(* IEC 61131-3 sources: StewartPlatform/Class/IONet, 1 file *)

(* ---- IONet.st ---- *)
(*!
<Class
	Name               = "IONet"
	Revision           = "0.0"
	RealtimeTask       = "false"
	CyclicTask         = "true"
	DefCyclictime      = "10 ms"
	BackgroundTask     = "false"
	Sigmatek           = "false"
	OSInterface        = "false"
	HighPriority       = "false"
	Automatic          = "false"
	UpdateMode         = "Prescan"
	SharedCommandTable = "true"
	Objectsize         = "(720,360)">
	<Channels>
		<Server Name="ClassSvr" Visualized="false" Initialize="false" WriteProtected="true" Retentive="false"/>
		<Server Name="Counter1" Visualized="false" Initialize="true" DefValue="2000" WriteProtected="false" Retentive="File"/>
		<Server Name="Counter2" Visualized="false" Initialize="true" DefValue="8000" WriteProtected="false" Retentive="File"/>
		<Server Name="Counter3" Visualized="false" Initialize="true" DefValue="5000" WriteProtected="false" Retentive="File"/>
		<Server Name="DefaultSpeed" Visualized="false" Initialize="false" WriteProtected="false" Retentive="File"/>
		<Server Name="diff" Visualized="false" Initialize="false" WriteProtected="false" Retentive="File"/>
		<Server Name="Direction1" Visualized="false" Initialize="true" DefValue="0" WriteProtected="false" Retentive="File"/>
		<Server Name="Direction2" Visualized="false" Initialize="true" DefValue="1" WriteProtected="false" Retentive="File"/>
		<Server Name="Direction3" Visualized="false" Initialize="true" DefValue="0" WriteProtected="false" Retentive="File"/>
		<Server Name="DropDownSpeed" Visualized="false" Initialize="false" WriteProtected="false" Retentive="File"/>
		<Server Name="Error1" Visualized="false" Initialize="false" WriteProtected="false" Retentive="File"/>
		<Server Name="Error2" Visualized="false" Initialize="false" WriteProtected="false" Retentive="File"/>
		<Server Name="Error3" Visualized="false" Initialize="false" WriteProtected="false" Retentive="File"/>
		<Server Name="Error4" Visualized="false" Initialize="false" WriteProtected="false" Retentive="File"/>
		<Server Name="Error5" Visualized="false" Initialize="false" WriteProtected="false" Retentive="File"/>
		<Server Name="Error6" Visualized="false" Initialize="false" WriteProtected="false" Retentive="File"/>
		<Server Name="InitCounter1" Visualized="false" Initialize="false" WriteProtected="false" Retentive="File"/>
		<Server Name="InitialTolerance" Visualized="false" Initialize="false" WriteProtected="false" Retentive="File"/>
		<Server Name="Integrator1" Visualized="false" Initialize="false" WriteProtected="false" Retentive="File"/>
		<Server Name="Integrator2" Visualized="false" Initialize="false" WriteProtected="false" Retentive="File"/>
		<Server Name="Integrator3" Visualized="false" Initialize="false" WriteProtected="false" Retentive="File"/>
		<Server Name="Integrator4" Visualized="false" Initialize="false" WriteProtected="false" Retentive="File"/>
		<Server Name="Integrator5" Visualized="false" Initialize="false" WriteProtected="false" Retentive="File"/>
		<Server Name="Integrator6" Visualized="false" Initialize="false" WriteProtected="false" Retentive="File"/>
		<Server Name="Kd" Visualized="false" Initialize="true" DefValue="0" WriteProtected="false" Retentive="File"/>
		<Server Name="Ki" Visualized="false" Initialize="false" WriteProtected="false" Retentive="File"/>
		<Server Name="Kp" Visualized="false" Initialize="true" DefValue="5" WriteProtected="false" Retentive="File"/>
		<Server Name="LowerLimit" Visualized="false" Initialize="false" WriteProtected="false" Retentive="File"/>
		<Server Name="Mode" Visualized="false" Initialize="false" WriteProtected="false" Retentive="File"/>
		<Server Name="ModeDoneCounter" Visualized="false" Initialize="false" WriteProtected="true" Retentive="false"/>
		<Server Name="ModeDoneSmoother" Visualized="false" Initialize="false" WriteProtected="false" Retentive="File"/>
		<Server Name="Phase" Visualized="false" Initialize="false" WriteProtected="false" Retentive="File"/>
		<Server Name="Prior_error1" Visualized="false" Initialize="false" WriteProtected="false" Retentive="File"/>
		<Server Name="Prior_error2" Visualized="false" Initialize="false" WriteProtected="false" Retentive="File"/>
		<Server Name="Prior_error3" Visualized="false" Initialize="false" WriteProtected="false" Retentive="File"/>
		<Server Name="Prior_error4" Visualized="false" Initialize="false" WriteProtected="false" Retentive="File"/>
		<Server Name="Prior_error5" Visualized="false" Initialize="false" WriteProtected="false" Retentive="File"/>
		<Server Name="Prior_error6" Visualized="false" Initialize="false" WriteProtected="false" Retentive="File"/>
		<Server Name="Speed" Visualized="false" Initialize="false" WriteProtected="false" Retentive="File"/>
		<Server Name="System_state" Visualized="false" Initialize="false" WriteProtected="false" Retentive="File"/>
		<Server Name="UpperLimit" Visualized="false" Initialize="false" WriteProtected="false" Retentive="File"/>
		<Client Name="EnableCircuit" Required="true" Internal="false"/>
		<Client Name="ExternalController" Required="true" Internal="false"/>
		<Client Name="I1" Required="true" Internal="false"/>
		<Client Name="I2" Required="true" Internal="false"/>
		<Client Name="I3" Required="true" Internal="false"/>
		<Client Name="I4" Required="true" Internal="false"/>
		<Client Name="I5" Required="true" Internal="false"/>
		<Client Name="I6" Required="true" Internal="false"/>
		<Client Name="O1" Required="true" Internal="false"/>
		<Client Name="O2" Required="true" Internal="false"/>
		<Client Name="O3" Required="true" Internal="false"/>
		<Client Name="O4" Required="true" Internal="false"/>
		<Client Name="O5" Required="true" Internal="false"/>
		<Client Name="O6" Required="true" Internal="false"/>
		<Client Name="Pressurize" Required="true" Internal="false"/>
		<Client Name="ResetButton" Required="true" Internal="false"/>
		<Client Name="ResetButtonLamp" Required="true" Internal="false"/>
		<Client Name="ResetEStop" Required="true" Internal="false"/>
		<Client Name="StartButton" Required="true" Internal="false"/>
		<Client Name="StartButtonLamp" Required="true" Internal="false"/>
		<Client Name="StartPumps" Required="true" Internal="false"/>
		<Client Name="StopButton" Required="true" Internal="false"/>
		<Client Name="StopButtonLamp" Required="true" Internal="false"/>
		<Client Name="SystemEnable" Required="true" Internal="false"/>
		<Client Name="SystemOKLamp" Required="true" Internal="false"/>
	</Channels>
</Class>
*)
IONet : CLASS
  //Servers:
	ClassSvr 	: SvrChCmd_DINT;
	Counter1 	: SvrCh_DINT;
	Counter2 	: SvrCh_DINT;
	Counter3 	: SvrCh_DINT;
	InitCounter1 	: SvrCh_DINT;
	Direction1 	: SvrCh_UDINT;
	Direction2 	: SvrCh_DINT;
	Direction3 	: SvrCh_DINT;
	Kp 	: SvrCh_DINT;
	Kd 	: SvrCh_DINT;
	Ki 	: SvrCh_DINT;
	Mode 	: SvrCh_DINT;
	Phase 	: SvrCh_DINT;
	System_state 	: SvrCh_DINT;
	Speed 	: SvrCh_DINT;
	DropDownSpeed 	: SvrCh_DINT;
	DefaultSpeed 	: SvrCh_DINT;
	Prior_error1 	: SvrCh_DINT;
	Prior_error2 	: SvrCh_DINT;
	Prior_error3 	: SvrCh_DINT;
	Prior_error4 	: SvrCh_DINT;
	Prior_error5 	: SvrCh_DINT;
	Prior_error6 	: SvrCh_DINT;
	Error1 	: SvrCh_DINT;
	Error2 	: SvrCh_DINT;
	Error3 	: SvrCh_DINT;
	Error4 	: SvrCh_DINT;
	Error5 	: SvrCh_DINT;
	Error6 	: SvrCh_DINT;
	Integrator1 	: SvrCh_DINT;
	Integrator2 	: SvrCh_DINT;
	Integrator3 	: SvrCh_DINT;
	Integrator4 	: SvrCh_DINT;
	Integrator5 	: SvrCh_DINT;
	Integrator6 	: SvrCh_DINT;
	LowerLimit 	: SvrCh_DINT;
	UpperLimit 	: SvrCh_DINT;
	diff 	: SvrCh_DINT;
	InitialTolerance 	: SvrCh_DINT;
	ModeDoneSmoother 	: SvrCh_DINT;
	ModeDoneCounter 	: SvrCh_DINT;
  //Clients:
	StartButton 	: CltCh_DINT;
	StartButtonLamp 	: CltCh_DINT;
	StopButton 	: CltCh_DINT;
	StopButtonLamp 	: CltCh_DINT;
	ResetButton 	: CltCh_DINT;
	ResetButtonLamp 	: CltCh_DINT;
	SystemEnable 	: CltCh_DINT;
	EnableCircuit 	: CltCh_DINT;
	SystemOKLamp 	: CltCh_DINT;
	StartPumps 	: CltCh_DINT;
	Pressurize 	: CltCh_DINT;
	ResetEStop 	: CltCh_DINT;
	ExternalController 	: CltCh_DINT;
	O1 	: CltCh_DINT;
	O2 	: CltCh_DINT;
	O3 	: CltCh_DINT;
	O4 	: CltCh_DINT;
	O5 	: CltCh_DINT;
	O6 	: CltCh_DINT;
	I1 	: CltCh_DINT;
	I2 	: CltCh_DINT;
	I3 	: CltCh_DINT;
	I4 	: CltCh_DINT;
	I5 	: CltCh_DINT;
	I6 	: CltCh_DINT;
  //Variables:
  //Functions:

	FUNCTION VIRTUAL GLOBAL Init;

	FUNCTION VIRTUAL GLOBAL CyWork
		VAR_INPUT
			EAX 	: UDINT;
		END_VAR
		VAR_OUTPUT
			state (EAX) 	: UDINT;
		END_VAR;

	FUNCTION LimitOutput
		VAR_INPUT
			unlimited_output 	: DINT;
		END_VAR
		VAR_OUTPUT
			limited_output 	: DINT;
		END_VAR;

	FUNCTION UpdateMode;

	FUNCTION InitializeCounters;

	FUNCTION UpdateCounters;

	FUNCTION DecreaseCounters;

	FUNCTION CylRef
		VAR_INPUT
			cyl 	: DINT;
		END_VAR
		VAR_OUTPUT
			ref 	: DINT;
		END_VAR;

	FUNCTION GoToInitial
		VAR_INPUT
			ref 	: DINT;
			actual 	: DINT;
		END_VAR
		VAR_OUTPUT
			newref 	: DINT;
		END_VAR;

	FUNCTION ResetPriorErrors;

	FUNCTION SetPriorErrors;

	FUNCTION ResetIntegrators;

	FUNCTION UpdateIntegrators;

	FUNCTION InitializeMode;

	FUNCTION AbsoluteValue
		VAR_INPUT
			Actual 	: DINT;
		END_VAR
		VAR_OUTPUT
			Absolute 	: DINT;
		END_VAR;
  //Tables:
	FUNCTION @STD
		VAR_OUTPUT
			ret_code	: CONFSTATES;
		END_VAR;
	FUNCTION GLOBAL TAB @CT_;
END_CLASS;

FUNCTION VIRTUAL GLOBAL IONet::Init
  if _FirstScan then
    Kp := 5;
    Kd := 20;
    Ki := 1;
    LowerLimit := 500;        // Lowest reachable point of cylinders
    Direction1 := 0;
    Direction2 := 0;
    Direction3 := 0;
    Counter1 := LowerLimit;
    Counter2 := LowerLimit;
    Counter3 := LowerLimit;
    DefaultSpeed := 6;        // Speed with which to increase counters every 10ms
    InitialTolerance := 300;  // Tolerance to initial mode position below which the mode is started
    DropDownSpeed := 10;      // Speed to drop down with when stop button is pressed
    System_state := 0;        // System state: 0 = SAFETY, 1 = ON, 2 = IDLE, 3 = PAUSED
    // SAFETY: a safety reset is required to go to System_state IDLE
    // ON: system is doing a sequence of movements
    // IDLE: System slowly moves to lowest position and stays there (controlled by buttons)
    // PAUSED: System slowly moves to lowest position and stays there (controlled by external controller)
    Mode := 1;                // Mode indicates which movement to perform
    ModeDoneSmoother := 50;   // To let the platform stabilize before starting next mode
    ModeDoneCounter := 0;
    Phase := 1;               // Phase indicates the part of the mode we are in (1 = go to initial, 2 = outbound, 3 = inbound, 4 = done)
    // Mode 1: up-down Z-direction (cylinder 1-6 use direction1 and counter1)
    // Mode 2: rotate yaw (cylinder 1,3,5 use direction1 and counter1, others use direction2 and counter2)
    // Mode 3: simultaneous roll-pitch (cylinder 1&6 use direction1 and counter1, cylinder 2&3 use direction2 and counter2, others use direction3 and counter3)
    // Mode 4: planar x-y direction TODO
    ResetPriorErrors();       // Reset prior errors for derivative control action
    ResetIntegrators();       // Reset integrators for integral control action
  end_if;

END_FUNCTION

FUNCTION VIRTUAL GLOBAL IONet::CyWork
	VAR_INPUT
		EAX 	: UDINT;
	END_VAR
	VAR_OUTPUT
		state (EAX) 	: UDINT;
	END_VAR

  // Read all inputs
	StartButton := StartButton.Read();
	StopButton := StopButton.Read();
	ResetButton := ResetButton.Read();
  SystemEnable := SystemEnable.Read(); // Safety circuit input
  ExternalController := ExternalController.Read(); // External controller
  I1 := I1.Read();
  I2 := I2.Read();
  I3 := I3.Read();
  I4 := I4.Read();
  I5 := I5.Read();
  I6 := I6.Read();

  // If safety circuit is OK, enable circuit and pumps
  // THIS CHECK SHOULD ALWAYS BE AT THE BEGINNING OF THE LOOP
  // ***************************************
  if SystemEnable = 1 then
    SystemOKLamp := 1;
    EnableCircuit := 1;
    StartPumps := 1;
    // TODO: pressure low should prevent system from falling down but this does not work currently
    Pressurize := 1; // no outwards cylinder movement when 0
  else
    // Set state variables
    System_state := 0;      // System state SAFETY
    Mode := 1;              // Mode starts at 1 again
    InitializeMode();       // Re-initialize mode
    ResetPriorErrors();     // Reset prior errors for derivative control action
    ResetIntegrators();     // Reset integrators for integral control action
    // Turn everything off
    ResetEStop := 0;
    SystemOKLamp := 0;
    EnableCircuit := 0;
    StartPumps := 0;
    Pressurize := 0;        // no outwards cylinder movement when 0
  end_if;

  // Handle inputs of stop and start button
  if StopButton = 1 then
    // StopButton (red) lets the system go to state 2 (IDLE), transition only possible from state 1 (ON) or state 3 (PAUSED)
    if System_state = 1 | System_state = 3 then
      // Stop state ON/PAUSED and go to state IDLE
      System_state := 2;
    end_if;
    // Otherwise this does nothing
  elsif ExternalController = 0 then
    // External controller low lets the system go to state 3 (PAUSED), transition only possible from state 1 (ON)
    if System_state = 1 then
      // Stop state ON and go to state PAUSED
      System_state := 3;
    end_if;
  elsif StartButton = 1 then
    // StartButton (green) lets the system go to state 1 (ON), transition only possible from state 2 (IDLE)
    if System_state = 2 then
      // Stop state IDLE and go to state ON
      System_state := 1;
      ResetPriorErrors();
      ResetIntegrators();
      Mode := 1;
      InitializeMode();
    end_if;
    // Otherwise this does nothing
  elsif ExternalController = 1 then
    // External controller high means that the system should move (state 2), transition only possible from state 3 (PAUSED)
    if System_state = 3 then
      // Stop state PAUSED and go to state ON
      System_state := 1;
      // ResetPriorErrors();
      // ResetIntegrators();
      // Mode := 1;
      // InitializeMode();
    end_if;
  end_if;

  // Provide feedback on the current system state
  if System_state = 0 then
    StartButtonLamp := 0;
    StopButtonLamp := 0;
    ResetButtonLamp := 1;
  elsif System_state = 1 then
    StartButtonLamp := 1;
    StopButtonLamp := 0;
    ResetButtonLamp := 0;
  elsif System_state = 2 then
    StartButtonLamp := 0;
    StopButtonLamp := 1;
    ResetButtonLamp := 0;
  elsif System_state = 3 then
    StartButtonLamp := 0;
    StopButtonLamp := 0;
    ResetButtonLamp := 0;
  end_if;

  // SYSTEM BEHAVIOR
  // State SAFETY: Do nothing (since we cannot control the cylinders anyway)
  if System_state = 0 then
    O1 := 0;
    O2 := 0;
    O3 := 0;
    O4 := 0;
    O5 := 0;
    O6 := 0;
  else
    // State IDLE: slowly move downwards
    if System_state = 2 then
      DecreaseCounters();
    // State ON: perform movements according to the current Mode
    elsif System_state = 1 then
      // If previous mode is done, update it
      if Phase = 4 then
        UpdateMode(); // Will also reset Phase to 1
      elsif Phase = 2 | Phase = 3 then
        // Update the references according to the mode movement
        UpdateCounters();
      end_if;
      // in Phase 1, counters do not have to be updated
    end_if;

    // Calculate errors
    Error1 := CylRef(cyl:=1)-I1;
    Error2 := CylRef(cyl:=2)-I2;
    Error3 := CylRef(cyl:=3)-I3;
    Error4 := CylRef(cyl:=4)-I4;
    Error5 := CylRef(cyl:=5)-I5;
    Error6 := CylRef(cyl:=6)-I6;

    if Phase = 1 then
      if AbsoluteValue(Actual:=Error1) < InitialTolerance & AbsoluteValue(Actual:=Error2) < InitialTolerance & AbsoluteValue(Actual:=Error3) < InitialTolerance & AbsoluteValue(Actual:=Error4) < InitialTolerance & AbsoluteValue(Actual:=Error5) < InitialTolerance & AbsoluteValue(Actual:=Error6) < InitialTolerance then
        // All cylinders are now close enough to their initial positions so we can enter Phase 2
        Phase := 2;
      end_if;
    end_if;

    // Update controller integrators
    UpdateIntegrators();
    // Apply controllers
    O1 := Error1*Kp + Integrator1*Ki + (Error1-Prior_error1)*1*Kd; // Note: multiplied by 1 instead of 100 to allow lower damping
    O2 := Error2*Kp + Integrator2*Ki + (Error2-Prior_error2)*1*Kd; // Note: multiplied by 1 instead of 100 to allow lower damping
    O3 := Error3*Kp + Integrator3*Ki + (Error3-Prior_error3)*1*Kd; // Note: multiplied by 1 instead of 100 to allow lower damping
    O4 := Error4*Kp + Integrator4*Ki + (Error4-Prior_error4)*1*Kd; // Note: multiplied by 1 instead of 100 to allow lower damping
    O5 := Error5*Kp + Integrator5*Ki + (Error5-Prior_error5)*1*Kd; // Note: multiplied by 1 instead of 100 to allow lower damping
    O6 := Error6*Kp + Integrator6*Ki + (Error6-Prior_error6)*1*Kd; // Note: multiplied by 1 instead of 100 to allow lower damping
    // Set prior errors for next iteration
    SetPriorErrors();
  end_if;

  // Limit the outputs to their maximum range
  O1 := LimitOutput(unlimited_output:=O1);
  O2 := LimitOutput(unlimited_output:=O2);
  O3 := LimitOutput(unlimited_output:=O3);
  O4 := LimitOutput(unlimited_output:=O4);
  O5 := LimitOutput(unlimited_output:=O5);
  O6 := LimitOutput(unlimited_output:=O6);

  // Pressing the ResetButton (blue) resets the safety circuit
  // SHOULD ALWAYS BE AT THE END OF THE LOOP
  // ***************************************
  if ResetButton = 1 then
    ResetEStop := 1;
    // Go to state 2 (IDLE) for now, if safety reset fails we go back to state 0 (SAFETY) anyway
    System_state := 2;
  end_if;

  // Write all outputs
  SystemOKLamp.Write(SystemOKLamp);
  EnableCircuit.Write(EnableCircuit);
  StartPumps.Write(StartPumps);
  Pressurize.Write(Pressurize);
  ResetEStop.Write(ResetEStop);
  StartButtonLamp.Write(StartButtonLamp);
  StopButtonLamp.Write(StopButtonLamp);
  ResetButtonLamp.Write(ResetButtonLamp);
  O1.Write(O1);
  O2.Write(O2);
  O3.Write(O3);
  O4.Write(O4);
  O5.Write(O5);
  O6.Write(O6);

  state := READY;

END_FUNCTION

// Saturate the outputs in range -10000 to +10000
FUNCTION IONet::LimitOutput
	VAR_INPUT
		unlimited_output 	: DINT;
	END_VAR
	VAR_OUTPUT
		limited_output 	: DINT;
	END_VAR

  if unlimited_output > 10000 then
    limited_output := 10000;
  elsif unlimited_output < -10000 then
    limited_output := -10000;
  else
    limited_output := unlimited_output;
  end_if;

END_FUNCTION

FUNCTION IONet::UpdateMode
  if mode >= 3 then
    Mode := 1;            // Go back to mode 1
  else
    Mode += 1;            // Go to next mode
  end_if;
  InitializeMode();
END_FUNCTION

FUNCTION IONet::InitializeMode
  Phase := 1;
  if mode = 1 | mode = 2 then
    UpperLimit := 9000;
    Speed := 2*DefaultSpeed;
  else
    UpperLimit := 5000;
    Speed := DefaultSpeed;
  end_if;
  InitializeCounters();
END_FUNCTION

FUNCTION IONet::InitializeCounters
  if Mode = 1 then
    Counter1 := LowerLimit;
    Direction1 := 0;
    Counter2 := LowerLimit;
    Direction2 := 0;
    Counter3 := LowerLimit;
    Direction3 := 0;
  elsif Mode = 2 then
    Counter1 := LowerLimit + (UpperLimit - LowerLimit)/2;
    Direction1 := 0;
    Counter2 := LowerLimit + (UpperLimit - LowerLimit)/2;
    Direction2 := 1;
    Counter3 := LowerLimit;
    Direction3 := 0;
  elsif Mode = 3 then
    Counter1 := LowerLimit + (UpperLimit - LowerLimit)/3*2;
    Direction1 := 0;
    Counter2 := LowerLimit + (UpperLimit - LowerLimit)/3;
    Direction2 := 0;
    Counter3 := LowerLimit + (UpperLimit - LowerLimit)/3;
    Direction3 := 1;
  else
    Counter1 := LowerLimit;
    Direction1 := 0;
    Counter2 := LowerLimit;
    Direction2 := 0;
    Counter3 := LowerLimit;
    Direction3 := 0;
  end_if;
  InitCounter1 := Counter1;
  ModeDoneCounter := 0;
END_FUNCTION

FUNCTION IONet::UpdateCounters
  // Direction 1 is in control of the Phase
  if Direction1 = 0 then
    Counter1 += Speed;
    if Phase = 3 & Counter1 >= InitCounter1 then
      if ModeDoneCounter >= ModeDoneSmoother then
        Phase := 4;  // To done phase
      else
        // Stabilize first for smooth switch to next mode
        ModeDoneCounter += 1;
        Counter1 -= Speed;
        return;
      end_if;
    elsif Counter1 >= UpperLimit then
      Direction1 := 1;
      Phase := 3; // To inbound movement phase
    end_if;
  else
    Counter1 -= Speed;
    if Counter1 <= LowerLimit then
      Direction1 := 0;
    end_if;
  end_if;
  if Direction2 = 0 then
    Counter2 += Speed;
    if Counter2 >= UpperLimit then
      Direction2 := 1;
    end_if;
  else
    Counter2 -= Speed;
    if Counter2 <= LowerLimit then
      Direction2 := 0;
    end_if;
  end_if;
  if Direction3 = 0 then
    Counter3 += Speed;
    if Counter3 >= UpperLimit then
      Direction3 := 1;
    end_if;
  else
    Counter3 -= Speed;
    if Counter3 <= LowerLimit then
      Direction3 := 0;
    end_if;
  end_if;
END_FUNCTION

FUNCTION IONet::DecreaseCounters
  Counter1 -= DropDownSpeed;
  if Counter1 < LowerLimit then
    Counter1 := LowerLimit;
  end_if;
  Counter2 -= DropDownSpeed;
  if Counter2 < LowerLimit then
    Counter2 := LowerLimit;
  end_if;
  Counter3 -= DropDownSpeed;
  if Counter3 < LowerLimit then
    Counter3 := LowerLimit;
  end_if;
END_FUNCTION

// Get the reference for a certain cylinder
FUNCTION IONet::CylRef
	VAR_INPUT
		cyl 	: DINT;
	END_VAR
	VAR_OUTPUT
		ref 	: DINT;
	END_VAR

  if mode = 1 then
    // All cylinders follow reference of Counter1
    ref := Counter1;
  elsif mode = 2 then
    // Cylinders 1, 3 and 5 follow reference of Counter1, others are follow Counter2
    case cyl of
      1: ref := Counter1;
      2: ref := Counter2;
      3: ref := Counter1;
      4: ref := Counter2;
      5: ref := Counter1;
      6: ref := Counter2;
    end_case;
  elsif mode = 3 then
    // Cylinders 3 and 4 follow reference of Counter1, others are 0
    case cyl of
      1: ref := Counter1;
      2: ref := Counter2;
      3: ref := Counter2;
      4: ref := Counter3;
      5: ref := Counter3;
      6: ref := Counter1;
    end_case;
  else
    // All cylinders follow reference of Counter1
    ref := Counter1;
  end_if;

  if Phase = 1 then
    if System_state = 3 then
      // Do nothing
      case cyl of
        1: ref := I1;
        2: ref := I2;
        3: ref := I3;
        4: ref := I4;
        5: ref := I5;
        6: ref := I6;
      end_case;
    else
      // First slowly move to initial position of cylinder
      case cyl of
        1: ref := GoToInitial(ref:=ref, actual:=I1);
        2: ref := GoToInitial(ref:=ref, actual:=I2);
        3: ref := GoToInitial(ref:=ref, actual:=I3);
        4: ref := GoToInitial(ref:=ref, actual:=I4);
        5: ref := GoToInitial(ref:=ref, actual:=I5);
        6: ref := GoToInitial(ref:=ref, actual:=I6);
      end_case;
    end_if;
  end_if;

END_FUNCTION

FUNCTION IONet::GoToInitial
	VAR_INPUT
		ref 	: DINT;
		actual 	: DINT;
	END_VAR
	VAR_OUTPUT
		newref 	: DINT;
	END_VAR

  diff := ref-actual;
  if abs(diff) > InitialTolerance then
    // Move to initial position with controlled speed
    if diff > 0 then
      newref := actual + InitialTolerance;
    else
      newref := actual - InitialTolerance;
    end_if;
  else
    // Initial position is within speed range
    newref := ref;
  end_if;
END_FUNCTION

FUNCTION IONet::ResetPriorErrors
  Prior_error1 := 0;        // Used for derivative control action on cylinder 1
  Prior_error2 := 0;        // Used for derivative control action on cylinder 2
  Prior_error3 := 0;        // Used for derivative control action on cylinder 3
  Prior_error4 := 0;        // Used for derivative control action on cylinder 4
  Prior_error5 := 0;        // Used for derivative control action on cylinder 5
  Prior_error6 := 0;        // Used for derivative control action on cylinder 6
END_FUNCTION

FUNCTION IONet::SetPriorErrors
  Prior_error1 := Error1;   // Used for derivative control action on cylinder 1
  Prior_error2 := Error2;   // Used for derivative control action on cylinder 2
  Prior_error3 := Error3;   // Used for derivative control action on cylinder 3
  Prior_error4 := Error4;   // Used for derivative control action on cylinder 4
  Prior_error5 := Error5;   // Used for derivative control action on cylinder 5
  Prior_error6 := Error6;   // Used for derivative control action on cylinder 6
END_FUNCTION

FUNCTION IONet::ResetIntegrators
  Integrator1 := 0;         // Used for integral control action on cylinder 1
  Integrator2 := 0;         // Used for integral control action on cylinder 2
  Integrator3 := 0;         // Used for integral control action on cylinder 3
  Integrator4 := 0;         // Used for integral control action on cylinder 4
  Integrator5 := 0;         // Used for integral control action on cylinder 5
  Integrator6 := 0;         // Used for integral control action on cylinder 6
END_FUNCTION

FUNCTION IONet::UpdateIntegrators
  Integrator1 += (Error1/100); // Note: divided by 100 because cycle time is 10ms
  Integrator2 += (Error2/100); // Note: divided by 100 because cycle time is 10ms
  Integrator3 += (Error3/100); // Note: divided by 100 because cycle time is 10ms
  Integrator4 += (Error4/100); // Note: divided by 100 because cycle time is 10ms
  Integrator5 += (Error5/100); // Note: divided by 100 because cycle time is 10ms
  Integrator6 += (Error6/100); // Note: divided by 100 because cycle time is 10ms
END_FUNCTION

FUNCTION IONet::AbsoluteValue
	VAR_INPUT
		Actual 	: DINT;
	END_VAR
	VAR_OUTPUT
		Absolute 	: DINT;
	END_VAR

  if Actual >= 0 then
    Absolute := Actual;
  else
    Absolute := -Actual;
  end_if;
END_FUNCTION
